PROGRAM MAIN
VAR
	fbTcpServer 	: FB_TcpServer;
	SrvNetId		: STRING := '';
	ServerAddress 	: STRING := '127.0.0.1';  //line specifies the IP address of the TCP server.
	ServerPort 		: UDINT := 2000;		  //specifies the port number of the TCP server.
	
	sResponse		: STRING;					//specifies the variable that will be used to send data to the TCP server.
	sCommand		: STRING;					//specifies the variable that will be used to receive data from the TCP server.
	bBusy			: BOOL;
	err				: BOOL;
	errid			: UDINT;
	
	Toggle 	: FB_Toggle;					 // toggle FB block for m0.0
	MemBit0 AT %MX0.0 : BOOL    := FALSE;    //memory bit to toggle and sent to client
	
END_VAR

fbTcpServer(
	NetId:= SrvNetId, 
	ServerAdr:= ServerAddress, 
	ServerPort:= ServerPort, 
	sSend := sResponse,
	sReceive=> sCommand, 
	bBusy=> bBusy, 
	err=> err, 
	errid=> errid);

Toggle(Timer:= T#500MS , Toggle_Out=> );		//FB_TOGGLE for MemBit0
MemBit0 := Toggle.Toggle_Out;

sResponse := sCommand;
IF sCommand = 'BIT-0' THEN
	IF MemBit0 THEN
		sResponse := '1';
	ELSE
		sResponse := '0';
	END_IF
END_IF

END_PROGRAM

(* stored: Version 1.1.0.1, ProductVersion 3.1.4024.6
   POU MAIN: Id {51edf94c-8a91-4167-a283-3931655e3d9d}, SpecialFunc None *)
